// TIA Portal V16 export
// export: Created 2021-07-12T14:47:20.4755064Z, ExportSetting WithDefaults, DisplayName Totally Integrated Automation Portal, DisplayVersion V16, DisplayName TIA Portal Version Control Interface, DisplayVersion V16, DisplayName TIA Portal Openness, DisplayVersion V16, DisplayName STEP 7 Professional, DisplayVersion V16, DisplayName STEP 7 Safety, DisplayVersion V16, DisplayName WinCC Professional, DisplayVersion V16
TYPE "SimaHydTO_typeHMIConnectionGetCharacteristicInterface"
TITLE = SimaHydTO_typeHMIConnectionGetCharacteristicInterface
// Function block interface of FB "GetCharacteristics"
// stored: IsFailsafeCompliant false
   STRUCT
      Command { S7_SetPoint := 'True'} : "SimaHydTO_typeHMIConnectionGetCharacteristicInterfaceCommand";   // HMI -> PLC: Commands to function block GetCharacteristics
      Status { S7_SetPoint := 'True'} : "SimaHydTO_typeHMIConnectionGetCharacteristicInterfaceStatus";   // PLC -> HMI: Status of function block GetCharacteristics
      ConfigData { S7_SetPoint := 'True'} : "LSimaHydTO_typeMeasurementConfig";
      MeasuredValues { S7_SetPoint := 'True'} : "LSimaHydTO_typeMeasuredValues";
   END_STRUCT;
END_TYPE
